ABB RobotStudio station: 6640_station_20220127-223635.rsstn

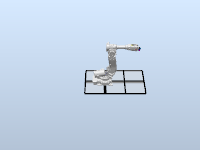
Station Station (saved by RobotStudio 21.4.9700.0)
Layout (positions relative to the parent item):
  - IRB6640_180_255__04 [mechanism, from Robots\IRB6640_180_255_G_04.rslib] at (0, 0, 0) mm; joint values [0, 0, 0, 0, 0.5236, 0] (rad or m)
